{attribute addProperty BoxType "ELM2644-0000-0016"}
{attribute addProperty Id "Outputs_Channel_3AT %Q*Outputs_Channel_E6FE5E20162"}
{attribute addProperty CRC "2151354313"}
{attribute addProperty SizeInBites "16"}
{attribute addProperty SizeInBytes "2"}
TYPE DO_Group_3_Outputs_803B0FC9 :
STRUCT
	{attribute addProperty Name "Outputs_Channel_3"}
	Outputs_Channel_3 AT %Q* : Outputs_Channel_E6FE5E20;
END_STRUCT
END_TYPE

(* stored: Version 1.2.0.0, ProductVersion 3.1.4024.9
   DUT DO_Group_3_Outputs_803B0FC9: Id {9f67b1ed-8516-4b1e-bd94-813b6a1fc96b} *)
